// TIA Portal project "Parcial_Segundo_Corte" (V16)

(* hardware
DEVICE "S71500/ET200MP station_2"  S7-1500 station
   slot 0: "PM 190W 120/230VAC"  PM 190W 120/230VAC  6EP1333-4BA00
   slot 0: "Perfil soporte_0"  Rack  6ES7 590-1***0-0AA0
   slot 1: "MAESTRO"  CPU 1516-3 PN/DP  6ES7 516-3AN02-0AB0  V2.8
      slot 3: "Display de la CPU_1"  6ES7591-1BA00-0AA0
      slot 32768: "Interfaz PROFINET_1"  X1
         slot 32769: "Puerto_1"  X1 P1
         slot 32770: "Puerto_2"  X1 P2
      slot 33024: "Interfaz PROFINET_2"  X2
         slot 33025: "Puerto_1"  X2 P1
      slot 33280: "Interfaz DP_1"  X3
      slot 34817: "Virtual CP interface port_1"  Virtual CP interface port  Virtual CP interface port
   slot 2: "DI 32x24VDC HF_1"  DI 32x24VDC HF  6ES7 521-1BL00-0AB0  V2.0
   slot 3: "DQ 32x24VDC/0.5A ST_1"  DQ 32x24VDC/0.5A ST  6ES7 522-1BL00-0AB0  V1.0
   slot 4: "AI 8xU/I/RTD/TC ST_1"  AI 8xU/I/RTD/TC ST  6ES7 531-7KF00-0AB0  V2.0
   slot 5: "AQ 4xU/I ST_1"  AQ 4xU/I ST  6ES7 532-5HD00-0AB0  V2.0
DEVICE "S71500/ET200MP station_1"  S7-1500 station
   slot 0: "Perfil soporte_0"  Rack  6ES7 590-1***0-0AA0
   slot 0: "PM 190W 120/230VAC"  PM 190W 120/230VAC  6EP1333-4BA00
   slot 1: "ESCLAVO"  CPU 1516-3 PN/DP  6ES7 516-3AN02-0AB0  V2.8
      slot 3: "Display de la CPU_1"  6ES7591-1BA00-0AA0
      slot 32768: "Interfaz PROFINET_1"  X1
         slot 32769: "Puerto_1"  X1 P1
         slot 32770: "Puerto_2"  X1 P2
      slot 33024: "Interfaz PROFINET_2"  X2
         slot 33025: "Puerto_1"  X2 P1
      slot 33280: "Interfaz DP_1"  X3
      slot 34817: "Virtual CP interface port_1"  Virtual CP interface port  Virtual CP interface port
   slot 2: "DI 32x24VDC HF_1"  DI 32x24VDC HF  6ES7 521-1BL00-0AB0  V2.0
   slot 3: "DQ 32x24VDC/0.5A ST_1"  DQ 32x24VDC/0.5A ST  6ES7 522-1BL00-0AB0  V1.0
   slot 4: "AI 8xU/I/RTD/TC ST_1"  AI 8xU/I/RTD/TC ST  6ES7 531-7KF00-0AB0  V2.0
   slot 5: "AQ 4xU/I ST_1"  AQ 4xU/I ST  6ES7 532-5HD00-0AB0  V2.0
DEVICE "S7300/ET200M station_2"  S7-300 station
   slot 0: "Perfil soporte_0"  Rail  6ES7 390-1***0-0AA0
   slot 1: "PS 307 5A_1"  PS 307 5A  6ES7 307-1EA00-0AA0
   slot 2: "ESCLAVO_300"  CPU 314C-2 DP  6ES7 314-6CG03-0AB0  V2.6
      slot 0: "Interfaz MPI_1"  X1
      slot 1: "Interfaz DP_1"  X2
      slot 2: "DI 24/DO 16_1"  DI24/DO16
      slot 3: "AI 5/AO 2_1"  AI5/AO2
      slot 4: "Contaje_1"  Counter
      slot 5: "Posicionamiento_1"  Positioning
DEVICE "S7300/ET200M station_1"  S7-300 station
   slot 0: "Perfil soporte_0"  Rail  6ES7 390-1***0-0AA0
   slot 1: "PS 307 5A_1"  PS 307 5A  6ES7 307-1EA00-0AA0
   slot 2: "MAESTRO_300"  CPU 314C-2 DP  6ES7 314-6CG03-0AB0  V2.6
      slot 0: "Interfaz MPI_1"  X1
      slot 1: "Interfaz DP_1"  X2
      slot 2: "DI 24/DO 16_1"  DI24/DO16
      slot 3: "AI 5/AO 2_1"  AI5/AO2
      slot 4: "Contaje_1"  Counter
      slot 5: "Posicionamiento_1"  Positioning
*)

// ===== PLC "ESCLAVO"  CPU 1516-3 PN/DP =====

VAR_GLOBAL   // PLC tag table "COMUNICACION"
   "Clock_Byte" AT %MB0 : Byte;
   "Clock_10Hz" AT %M0.0 : Bool;
   "Clock_5Hz" AT %M0.1 : Bool;
   "Clock_2.5Hz" AT %M0.2 : Bool;
   "Clock_2Hz" AT %M0.3 : Bool;
   "Clock_1.25Hz" AT %M0.4 : Bool;
   "Clock_1Hz" AT %M0.5 : Bool;
   "Clock_0.625Hz" AT %M0.6 : Bool;
   "Clock_0.5Hz" AT %M0.7 : Bool;
   "Tag_1" AT %MB30 : Byte;
   "Tag_2" AT %MB40 : Byte;
   "MARCAM30.0" AT %M30.0 : Bool;
   "MARCAM30.1" AT %M30.1 : Bool;
   "MARCAM30.2" AT %M30.2 : Bool;
   "MARCAM30.3" AT %M30.3 : Bool;
   "MARCAM30.4" AT %M30.4 : Bool;
   "MARCAM30.5" AT %M30.5 : Bool;
   "MARCAM30.6" AT %M30.6 : Bool;
   "MARCAM30.7" AT %M30.7 : Bool;
   "MARCAM40.0" AT %M40.0 : Bool;
   "MARCAM40.1" AT %M40.1 : Bool;
   "MARCAM40.2" AT %M40.2 : Bool;
   "MARCAM40.3" AT %M40.3 : Bool;
   "MARCAM40.4" AT %M40.4 : Bool;
   "MARCAM40.5" AT %M40.5 : Bool;
   "MARCAM40.6" AT %M40.6 : Bool;
   "MARCAM40.7" AT %M40.7 : Bool;
   "Tag_3" AT %M200.0 : Bool;
   "Tag_4" AT %M200.1 : Bool;
   "Tag_5" AT %M200.2 : Bool;
   "Tag_6" AT %M200.3 : Bool;
   "Tag_7" AT %M200.4 : Bool;
   "Tag_8" AT %M200.5 : Bool;
   "Tag_9" AT %M200.6 : Bool;
   "Tag_10" AT %M200.7 : Bool;
   "Tag_11" AT %M300.0 : Bool;
   "Tag_12" AT %M300.1 : Bool;
   "Tag_13" AT %M300.2 : Bool;
   "Tag_14" AT %M300.4 : Bool;
   "Tag_15" AT %M300.3 : Bool;
   "Tag_16" AT %M300.5 : Bool;
   "Tag_17" AT %M300.6 : Bool;
   "Tag_18" AT %M300.7 : Bool;
END_VAR

// folder: System blocks/Program resources

DATA_BLOCK "ESCLAVO_Receive_DB"   // DB2
{ S7_Optimized_Access := 'TRUE' }
AUTHOR : SIMATIC
FAMILY : MC7Plus
NAME : TC_IP_v4
VERSION : 1.0
// stored: InstanceOfName TCON_IP_v4
"TCON_IP_v4"
BEGIN
   ID := 1;
   InterfaceId := 64;
   LocalPort := 2000;
   RemoteAddress.ADDR[1] := 192;
   RemoteAddress.ADDR[2] := 168;
   RemoteAddress.ADDR[4] := 10;
END_DATA_BLOCK

// folder: (top level)

FUNCTION "comunicacion" : Void   // FC1, LAD
{ S7_Optimized_Access := 'TRUE' }
VERSION : 0.1
BEGIN

REGION Network 1: RECIBIR ESCLAVO
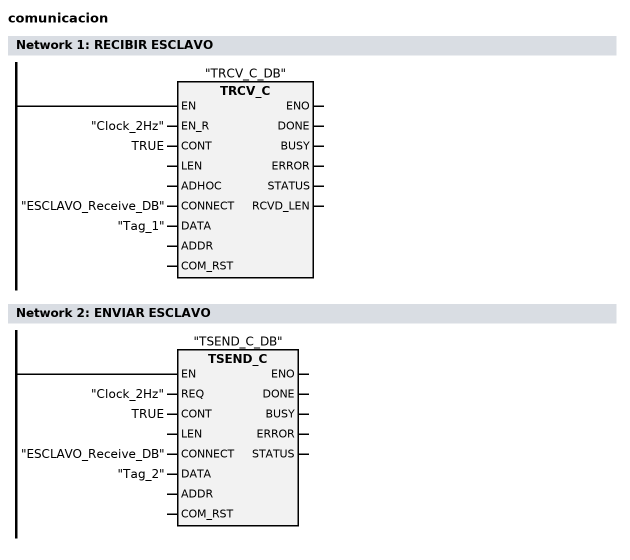
   "TRCV_C_DB"(EN_R := "Clock_2Hz", CONT := TRUE, CONNECT := "ESCLAVO_Receive_DB", DATA := "Tag_1");   // TRCV_C
END_REGION

REGION Network 2: ENVIAR ESCLAVO
   "TSEND_C_DB"(REQ := "Clock_2Hz", CONT := TRUE, CONNECT := "ESCLAVO_Receive_DB", DATA := "Tag_2");   // TSEND_C
END_REGION
END_FUNCTION

FUNCTION "compuertas" : Void   // FC2, LAD
{ S7_Optimized_Access := 'TRUE' }
VERSION : 0.1
BEGIN

REGION Network 1: SALIDAS ESCLAVO
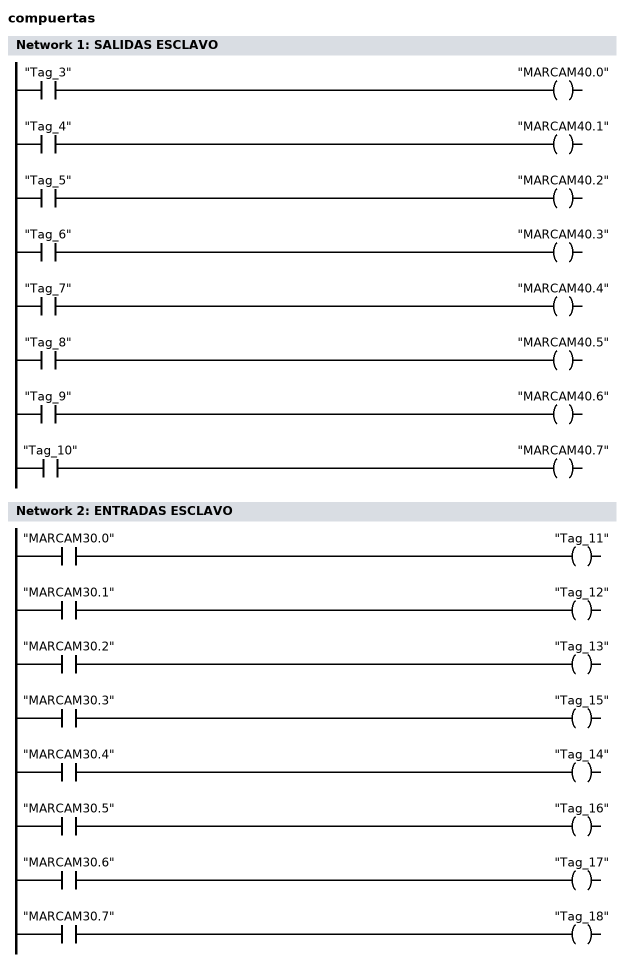
   RUNG wire#powerrail
      Contact( "Tag_3" )
      Coil( "MARCAM40.0" )
   END_RUNG
   RUNG wire#powerrail
      Contact( "Tag_4" )
      Coil( "MARCAM40.1" )
   END_RUNG
   RUNG wire#powerrail
      Contact( "Tag_5" )
      Coil( "MARCAM40.2" )
   END_RUNG
   RUNG wire#powerrail
      Contact( "Tag_6" )
      Coil( "MARCAM40.3" )
   END_RUNG
   RUNG wire#powerrail
      Contact( "Tag_7" )
      Coil( "MARCAM40.4" )
   END_RUNG
   RUNG wire#powerrail
      Contact( "Tag_8" )
      Coil( "MARCAM40.5" )
   END_RUNG
   RUNG wire#powerrail
      Contact( "Tag_9" )
      Coil( "MARCAM40.6" )
   END_RUNG
   RUNG wire#powerrail
      Contact( "Tag_10" )
      Coil( "MARCAM40.7" )
   END_RUNG
   // the same network as SCL:
   "MARCAM40.0" := "Tag_3";
   "MARCAM40.1" := "Tag_4";
   "MARCAM40.2" := "Tag_5";
   "MARCAM40.3" := "Tag_6";
   "MARCAM40.4" := "Tag_7";
   "MARCAM40.5" := "Tag_8";
   "MARCAM40.6" := "Tag_9";
   "MARCAM40.7" := "Tag_10";
END_REGION

REGION Network 2: ENTRADAS ESCLAVO
   RUNG wire#powerrail
      Contact( "MARCAM30.0" )
      Coil( "Tag_11" )
   END_RUNG
   RUNG wire#powerrail
      Contact( "MARCAM30.1" )
      Coil( "Tag_12" )
   END_RUNG
   RUNG wire#powerrail
      Contact( "MARCAM30.2" )
      Coil( "Tag_13" )
   END_RUNG
   RUNG wire#powerrail
      Contact( "MARCAM30.3" )
      Coil( "Tag_15" )
   END_RUNG
   RUNG wire#powerrail
      Contact( "MARCAM30.4" )
      Coil( "Tag_14" )
   END_RUNG
   RUNG wire#powerrail
      Contact( "MARCAM30.5" )
      Coil( "Tag_16" )
   END_RUNG
   RUNG wire#powerrail
      Contact( "MARCAM30.6" )
      Coil( "Tag_17" )
   END_RUNG
   RUNG wire#powerrail
      Contact( "MARCAM30.7" )
      Coil( "Tag_18" )
   END_RUNG
   // the same network as SCL:
   "Tag_11" := "MARCAM30.0";
   "Tag_12" := "MARCAM30.1";
   "Tag_13" := "MARCAM30.2";
   "Tag_15" := "MARCAM30.3";
   "Tag_14" := "MARCAM30.4";
   "Tag_16" := "MARCAM30.5";
   "Tag_17" := "MARCAM30.6";
   "Tag_18" := "MARCAM30.7";
END_REGION
END_FUNCTION

ORGANIZATION_BLOCK "Main"   // OB1, LAD, ProgramCycle
TITLE = "Main Program Sweep (Cycle)"
{ S7_Optimized_Access := 'TRUE' }
VERSION : 0.1
   VAR_INPUT
      Initial_Call : Bool;   // Initial call of this OB
      Remanence : Bool;   // =True, if remanent data are available
   END_VAR
BEGIN

REGION Network 1: COMUNICACION ETHERNET
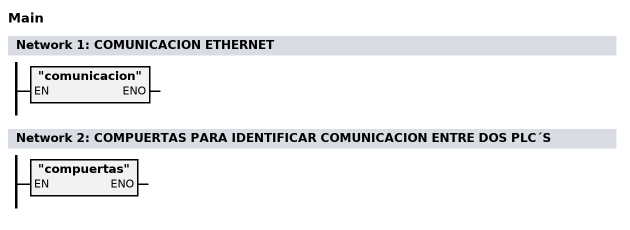
   RUNG wire#powerrail
      "comunicacion"()
   END_RUNG
   // the same network as SCL:
   "comunicacion"();
END_REGION

REGION Network 2: COMPUERTAS PARA IDENTIFICAR COMUNICACION ENTRE DOS PLC´S
   RUNG wire#powerrail
      "compuertas"()
   END_RUNG
   // the same network as SCL:
   "compuertas"();
END_REGION
END_ORGANIZATION_BLOCK

// ===== PLC "MAESTRO"  CPU 1516-3 PN/DP =====

VAR_GLOBAL   // PLC tag table "COMUNICACION"
   "Clock_Byte" AT %MB0 : Byte;
   "Clock_10Hz" AT %M0.0 : Bool;
   "Clock_5Hz" AT %M0.1 : Bool;
   "Clock_2.5Hz" AT %M0.2 : Bool;
   "Clock_2Hz" AT %M0.3 : Bool;
   "Clock_1.25Hz" AT %M0.4 : Bool;
   "Clock_1Hz" AT %M0.5 : Bool;
   "Clock_0.625Hz" AT %M0.6 : Bool;
   "Clock_0.5Hz" AT %M0.7 : Bool;
   "Tag_1" AT %MB20 : Byte;
   "Tag_2" AT %MB50 : Byte;
   "MARCAM20.0" AT %M20.0 : Bool;
   "MARCAM20.1" AT %M20.1 : Bool;
   "MARCAM20.2" AT %M20.2 : Bool;
   "MARCAM20.3" AT %M20.3 : Bool;
   "MARCAM20.4" AT %M20.4 : Bool;
   "MARCAM20.5" AT %M20.5 : Bool;
   "MARCAM20.6" AT %M20.6 : Bool;
   "MARCAM20.7" AT %M20.7 : Bool;
   "MARCAM50.0" AT %M50.0 : Bool;
   "MARCAM50.1" AT %M50.1 : Bool;
   "MARCAM50.2" AT %M50.2 : Bool;
   "MARCAM50.3" AT %M50.3 : Bool;
   "MARCAM50.4" AT %M50.4 : Bool;
   "MARCAM50.5" AT %M50.5 : Bool;
   "MARCAM50.6" AT %M50.6 : Bool;
   "MARCAM50.7" AT %M50.7 : Bool;
   "Tag_3" AT %M100.0 : Bool;
   "Tag_4" AT %M100.1 : Bool;
   "Tag_5" AT %M100.2 : Bool;
   "Tag_6" AT %M100.3 : Bool;
   "Tag_7" AT %M100.4 : Bool;
   "Tag_8" AT %M100.5 : Bool;
   "Tag_9" AT %M100.6 : Bool;
   "Tag_10" AT %M100.7 : Bool;
   "Tag_11" AT %M300.0 : Bool;
   "Tag_12" AT %M300.1 : Bool;
   "Tag_13" AT %M300.2 : Bool;
   "Tag_14" AT %M300.3 : Bool;
   "Tag_15" AT %M300.4 : Bool;
   "Tag_16" AT %M300.5 : Bool;
   "Tag_17" AT %M300.6 : Bool;
   "Tag_18" AT %M300.7 : Bool;
END_VAR

// folder: System blocks/Program resources

DATA_BLOCK "MAESTRO_Send_DB"   // DB2
{ S7_Optimized_Access := 'TRUE' }
AUTHOR : SIMATIC
FAMILY : MC7Plus
NAME : TC_IP_v4
VERSION : 1.0
// stored: InstanceOfName TCON_IP_v4
"TCON_IP_v4"
BEGIN
   ID := 1;
   InterfaceId := 64;
   RemotePort := 2000;
   ActiveEstablished := true;
   RemoteAddress.ADDR[1] := 192;
   RemoteAddress.ADDR[2] := 168;
   RemoteAddress.ADDR[4] := 20;
END_DATA_BLOCK

// folder: (top level)

FUNCTION "comunicacion" : Void   // FC1, LAD
{ S7_Optimized_Access := 'TRUE' }
VERSION : 0.1
BEGIN

REGION Network 1: ENVIAR MAESTRO
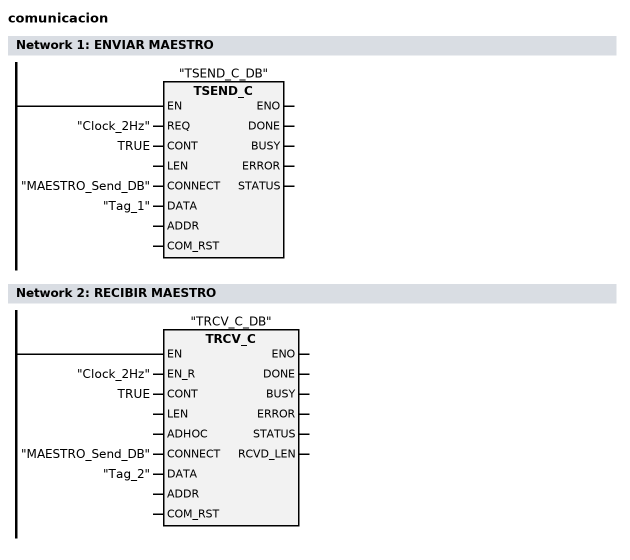
   "TSEND_C_DB"(REQ := "Clock_2Hz", CONT := TRUE, CONNECT := "MAESTRO_Send_DB", DATA := "Tag_1");   // TSEND_C
END_REGION

REGION Network 2: RECIBIR MAESTRO
   "TRCV_C_DB"(EN_R := "Clock_2Hz", CONT := TRUE, CONNECT := "MAESTRO_Send_DB", DATA := "Tag_2");   // TRCV_C
END_REGION
END_FUNCTION

FUNCTION "Compuertas" : Void   // FC2, LAD
{ S7_Optimized_Access := 'TRUE' }
VERSION : 0.1
BEGIN

REGION Network 1: SALIDAS MAESTRO
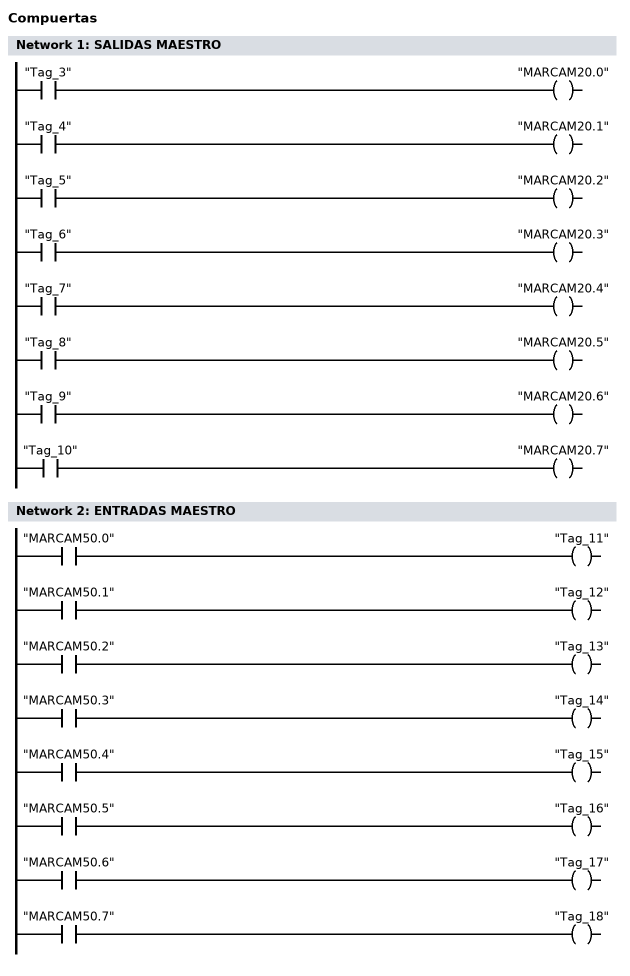
   RUNG wire#powerrail
      Contact( "Tag_3" )
      Coil( "MARCAM20.0" )
   END_RUNG
   RUNG wire#powerrail
      Contact( "Tag_4" )
      Coil( "MARCAM20.1" )
   END_RUNG
   RUNG wire#powerrail
      Contact( "Tag_5" )
      Coil( "MARCAM20.2" )
   END_RUNG
   RUNG wire#powerrail
      Contact( "Tag_6" )
      Coil( "MARCAM20.3" )
   END_RUNG
   RUNG wire#powerrail
      Contact( "Tag_7" )
      Coil( "MARCAM20.4" )
   END_RUNG
   RUNG wire#powerrail
      Contact( "Tag_8" )
      Coil( "MARCAM20.5" )
   END_RUNG
   RUNG wire#powerrail
      Contact( "Tag_9" )
      Coil( "MARCAM20.6" )
   END_RUNG
   RUNG wire#powerrail
      Contact( "Tag_10" )
      Coil( "MARCAM20.7" )
   END_RUNG
   // the same network as SCL:
   "MARCAM20.0" := "Tag_3";
   "MARCAM20.1" := "Tag_4";
   "MARCAM20.2" := "Tag_5";
   "MARCAM20.3" := "Tag_6";
   "MARCAM20.4" := "Tag_7";
   "MARCAM20.5" := "Tag_8";
   "MARCAM20.6" := "Tag_9";
   "MARCAM20.7" := "Tag_10";
END_REGION

REGION Network 2: ENTRADAS MAESTRO
   RUNG wire#powerrail
      Contact( "MARCAM50.0" )
      Coil( "Tag_11" )
   END_RUNG
   RUNG wire#powerrail
      Contact( "MARCAM50.1" )
      Coil( "Tag_12" )
   END_RUNG
   RUNG wire#powerrail
      Contact( "MARCAM50.2" )
      Coil( "Tag_13" )
   END_RUNG
   RUNG wire#powerrail
      Contact( "MARCAM50.3" )
      Coil( "Tag_14" )
   END_RUNG
   RUNG wire#powerrail
      Contact( "MARCAM50.4" )
      Coil( "Tag_15" )
   END_RUNG
   RUNG wire#powerrail
      Contact( "MARCAM50.5" )
      Coil( "Tag_16" )
   END_RUNG
   RUNG wire#powerrail
      Contact( "MARCAM50.6" )
      Coil( "Tag_17" )
   END_RUNG
   RUNG wire#powerrail
      Contact( "MARCAM50.7" )
      Coil( "Tag_18" )
   END_RUNG
   // the same network as SCL:
   "Tag_11" := "MARCAM50.0";
   "Tag_12" := "MARCAM50.1";
   "Tag_13" := "MARCAM50.2";
   "Tag_14" := "MARCAM50.3";
   "Tag_15" := "MARCAM50.4";
   "Tag_16" := "MARCAM50.5";
   "Tag_17" := "MARCAM50.6";
   "Tag_18" := "MARCAM50.7";
END_REGION
END_FUNCTION

ORGANIZATION_BLOCK "Main"   // OB1, LAD, ProgramCycle
TITLE = "Main Program Sweep (Cycle)"
{ S7_Optimized_Access := 'TRUE' }
VERSION : 0.1
   VAR_INPUT
      Initial_Call : Bool;   // Initial call of this OB
      Remanence : Bool;   // =True, if remanent data are available
   END_VAR
BEGIN

REGION Network 1
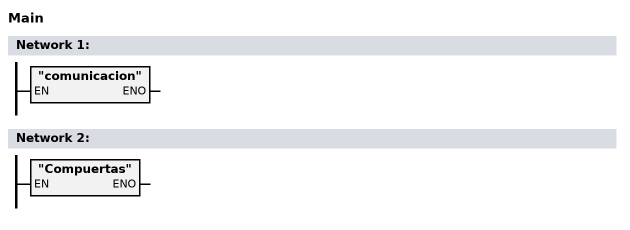
   RUNG wire#powerrail
      "comunicacion"()
   END_RUNG
   // the same network as SCL:
   "comunicacion"();
END_REGION

REGION Network 2
   RUNG wire#powerrail
      "Compuertas"()
   END_RUNG
   // the same network as SCL:
   "Compuertas"();
END_REGION
END_ORGANIZATION_BLOCK

// ===== PLC "MAESTRO_300"  CPU 314C-2 DP =====

VAR_GLOBAL   // PLC tag table "Tabla de variables estándar"
   "ENVIAR_DATO" AT %MB0 : Byte;
   "DATO_ENVIADO" AT %QB120 : Byte;
   "DATO_RECIBIDO" AT %IB240 : Byte;
   "VISUALIZAR_DATO" AT %MB3 : Byte;
END_VAR

FUNCTION "comunicacion" : Void   // FC1, LAD
{ S7_Optimized_Access := 'FALSE' }
VERSION : 0.1
BEGIN

REGION Network 1
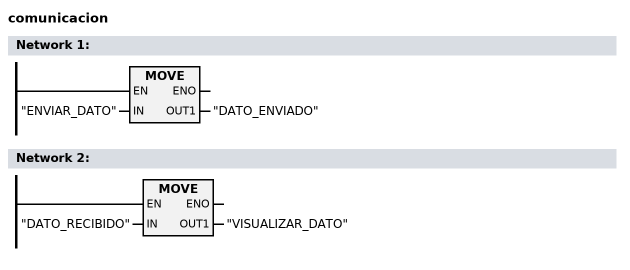
   RUNG wire#powerrail
      { S7_GenerateENO := "TRUE" } Move(in := "ENVIAR_DATO", out1 => "DATO_ENVIADO")
   END_RUNG
   // the same network as SCL:
   "DATO_ENVIADO" := "ENVIAR_DATO";
END_REGION

REGION Network 2
   RUNG wire#powerrail
      { S7_GenerateENO := "TRUE" } Move(in := "DATO_RECIBIDO", out1 => "VISUALIZAR_DATO")
   END_RUNG
   // the same network as SCL:
   "VISUALIZAR_DATO" := "DATO_RECIBIDO";
END_REGION
END_FUNCTION

ORGANIZATION_BLOCK "Main"   // OB1, LAD
TITLE = "Main Program Sweep (Cycle)"
{ S7_Optimized_Access := 'FALSE' }
VERSION : 0.1
   VAR_TEMP
      OB1_EV_CLASS : Byte;   // Bits 0-3 = 1 (Coming event), Bits 4-7 = 1 (Event class 1)
      OB1_SCAN_1 : Byte;   // 1 (Cold restart scan 1 of OB 1), 3 (Scan 2-n of OB 1)
      OB1_PRIORITY : Byte;   // Priority of OB Execution
      OB1_OB_NUMBR : Byte;   // 1 (Organization block 1, OB1)
      OB1_RESERVED_1 : Byte;   // Reserved for system
      OB1_RESERVED_2 : Byte;   // Reserved for system
      OB1_PREV_CYCLE : Int;   // Cycle time of previous OB1 scan (milliseconds)
      OB1_MIN_CYCLE : Int;   // Minimum cycle time of OB1 (milliseconds)
      OB1_MAX_CYCLE : Int;   // Maximum cycle time of OB1 (milliseconds)
      OB1_DATE_TIME : Date_And_Time;   // Date and time OB1 started
   END_VAR
BEGIN

REGION Network 1
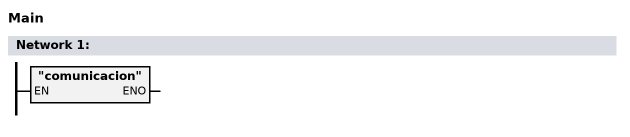
   RUNG wire#powerrail
      "comunicacion"()
   END_RUNG
   // the same network as SCL:
   "comunicacion"();
END_REGION
END_ORGANIZATION_BLOCK

ORGANIZATION_BLOCK "I/O_FLT1"   // OB82, FBD
TITLE = "I/O Point Fault"
{ S7_Optimized_Access := 'FALSE' }
VERSION : 0.1
   VAR_TEMP
      OB82_EV_CLASS : Byte;   // 16#39, Event class 3, Entering event state, Internal fault event
      OB82_FLT_ID : Byte;   // 16#XX, Fault identifcation code
      OB82_PRIORITY : Byte;   // Priority of OB Execution
      OB82_OB_NUMBR : Byte;   // 82 (Organization block 82, OB82)
      OB82_RESERVED_1 : Byte;   // Reserved for system
      OB82_IO_FLAG : Byte;   // Input (01010100), Output (01010101)
      OB82_MDL_ADDR : Word;   // Base address of module with fault
      OB82_MDL_DEFECT : Bool;   // Module defective
      OB82_INT_FAULT : Bool;   // Internal fault
      OB82_EXT_FAULT : Bool;   // External fault
      OB82_PNT_INFO : Bool;   // Point information
      OB82_EXT_VOLTAGE : Bool;   // External voltage low
      OB82_FLD_CONNCTR : Bool;   // Field wiring connector missing
      OB82_NO_CONFIG : Bool;   // Module has no configuration data
      OB82_CONFIG_ERR : Bool;   // Module has configuration error
      OB82_MDL_TYPE : Byte;   // Type of module
      OB82_SUB_MDL_ERR : Bool;   // Sub-Module is missing or has error
      OB82_COMM_FAULT : Bool;   // Communication fault
      OB82_MDL_STOP : Bool;   // Module is stopped
      OB82_WTCH_DOG_FLT : Bool;   // Watch dog timer stopped module
      OB82_INT_PS_FLT : Bool;   // Internal power supply fault
      OB82_PRIM_BATT_FLT : Bool;   // Primary battery is in fault
      OB82_BCKUP_BATT_FLT : Bool;   // Backup battery is in fault
      OB82_RESERVED_2 : Bool;   // Reserved for system
      OB82_RACK_FLT : Bool;   // Rack fault, only for bus interface module
      OB82_PROC_FLT : Bool;   // Processor fault
      OB82_EPROM_FLT : Bool;   // EPROM fault
      OB82_RAM_FLT : Bool;   // RAM fault
      OB82_ADU_FLT : Bool;   // ADU fault
      OB82_FUSE_FLT : Bool;   // Fuse fault
      OB82_HW_INTR_FLT : Bool;   // Hardware interupt input in fault
      OB82_RESERVED_3 : Bool;   // Reserved for system
      OB82_DATE_TIME : Date_And_Time;   // Date and time OB82 started
   END_VAR
BEGIN
END_ORGANIZATION_BLOCK

ORGANIZATION_BLOCK "RACK_FLT"   // OB86, FBD
TITLE = "Loss Of Rack Fault"
{ S7_Optimized_Access := 'FALSE' }
VERSION : 0.1
   VAR_TEMP
      OB86_EV_CLASS : Byte;   // 16#38/39 Event class 3
      OB86_FLT_ID : Byte;   // 16#C1/C4/C5, Fault identification code
      OB86_PRIORITY : Byte;   // Priority of OB Execution
      OB86_OB_NUMBR : Byte;   // 86 (Organization block 86, OB86)
      OB86_RESERVED_1 : Byte;   // Reserved for system
      OB86_RESERVED_2 : Byte;   // Reserved for system
      OB86_MDL_ADDR : Word;   // Base address of IM module in rack with fault
      OB86_RACKS_FLTD : Array[0..31] of Bool;   // Racks in fault
      OB86_DATE_TIME : Date_And_Time;   // Date and time OB86 started
   END_VAR
BEGIN
END_ORGANIZATION_BLOCK

// ===== PLC "ESCLAVO_300"  CPU 314C-2 DP =====

VAR_GLOBAL   // PLC tag table "Tabla de variables estándar"
   "ENVIAR_DATO" AT %MB0 : Byte;
   "DATO_ENVIADO" AT %QB240 : Byte;
   "DATO_RECIBIDO" AT %IB120 : Byte;
   "VISUALIZAR_DATO" AT %MB4 : Byte;
END_VAR

FUNCTION "comunicacion" : Void   // FC1, LAD
{ S7_Optimized_Access := 'FALSE' }
VERSION : 0.1
BEGIN

REGION Network 1
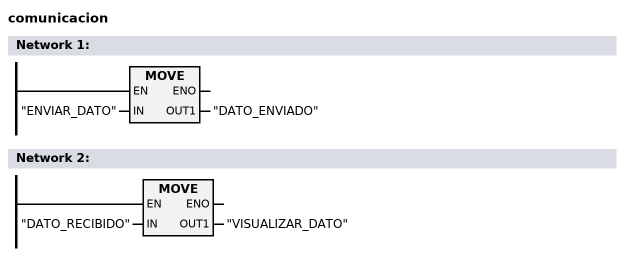
   RUNG wire#powerrail
      { S7_GenerateENO := "TRUE" } Move(in := "ENVIAR_DATO", out1 => "DATO_ENVIADO")
   END_RUNG
   // the same network as SCL:
   "DATO_ENVIADO" := "ENVIAR_DATO";
END_REGION

REGION Network 2
   RUNG wire#powerrail
      { S7_GenerateENO := "TRUE" } Move(in := "DATO_RECIBIDO", out1 => "VISUALIZAR_DATO")
   END_RUNG
   // the same network as SCL:
   "VISUALIZAR_DATO" := "DATO_RECIBIDO";
END_REGION
END_FUNCTION

ORGANIZATION_BLOCK "Main"   // OB1, LAD
TITLE = "Main Program Sweep (Cycle)"
{ S7_Optimized_Access := 'FALSE' }
VERSION : 0.1
   VAR_TEMP
      OB1_EV_CLASS : Byte;   // Bits 0-3 = 1 (Coming event), Bits 4-7 = 1 (Event class 1)
      OB1_SCAN_1 : Byte;   // 1 (Cold restart scan 1 of OB 1), 3 (Scan 2-n of OB 1)
      OB1_PRIORITY : Byte;   // Priority of OB Execution
      OB1_OB_NUMBR : Byte;   // 1 (Organization block 1, OB1)
      OB1_RESERVED_1 : Byte;   // Reserved for system
      OB1_RESERVED_2 : Byte;   // Reserved for system
      OB1_PREV_CYCLE : Int;   // Cycle time of previous OB1 scan (milliseconds)
      OB1_MIN_CYCLE : Int;   // Minimum cycle time of OB1 (milliseconds)
      OB1_MAX_CYCLE : Int;   // Maximum cycle time of OB1 (milliseconds)
      OB1_DATE_TIME : Date_And_Time;   // Date and time OB1 started
   END_VAR
BEGIN

REGION Network 1
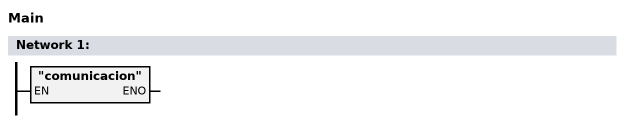
   RUNG wire#powerrail
      "comunicacion"()
   END_RUNG
   // the same network as SCL:
   "comunicacion"();
END_REGION
END_ORGANIZATION_BLOCK

ORGANIZATION_BLOCK "I/O_FLT1"   // OB82, FBD
TITLE = "I/O Point Fault"
{ S7_Optimized_Access := 'FALSE' }
VERSION : 0.1
   VAR_TEMP
      OB82_EV_CLASS : Byte;   // 16#39, Event class 3, Entering event state, Internal fault event
      OB82_FLT_ID : Byte;   // 16#XX, Fault identifcation code
      OB82_PRIORITY : Byte;   // Priority of OB Execution
      OB82_OB_NUMBR : Byte;   // 82 (Organization block 82, OB82)
      OB82_RESERVED_1 : Byte;   // Reserved for system
      OB82_IO_FLAG : Byte;   // Input (01010100), Output (01010101)
      OB82_MDL_ADDR : Word;   // Base address of module with fault
      OB82_MDL_DEFECT : Bool;   // Module defective
      OB82_INT_FAULT : Bool;   // Internal fault
      OB82_EXT_FAULT : Bool;   // External fault
      OB82_PNT_INFO : Bool;   // Point information
      OB82_EXT_VOLTAGE : Bool;   // External voltage low
      OB82_FLD_CONNCTR : Bool;   // Field wiring connector missing
      OB82_NO_CONFIG : Bool;   // Module has no configuration data
      OB82_CONFIG_ERR : Bool;   // Module has configuration error
      OB82_MDL_TYPE : Byte;   // Type of module
      OB82_SUB_MDL_ERR : Bool;   // Sub-Module is missing or has error
      OB82_COMM_FAULT : Bool;   // Communication fault
      OB82_MDL_STOP : Bool;   // Module is stopped
      OB82_WTCH_DOG_FLT : Bool;   // Watch dog timer stopped module
      OB82_INT_PS_FLT : Bool;   // Internal power supply fault
      OB82_PRIM_BATT_FLT : Bool;   // Primary battery is in fault
      OB82_BCKUP_BATT_FLT : Bool;   // Backup battery is in fault
      OB82_RESERVED_2 : Bool;   // Reserved for system
      OB82_RACK_FLT : Bool;   // Rack fault, only for bus interface module
      OB82_PROC_FLT : Bool;   // Processor fault
      OB82_EPROM_FLT : Bool;   // EPROM fault
      OB82_RAM_FLT : Bool;   // RAM fault
      OB82_ADU_FLT : Bool;   // ADU fault
      OB82_FUSE_FLT : Bool;   // Fuse fault
      OB82_HW_INTR_FLT : Bool;   // Hardware interupt input in fault
      OB82_RESERVED_3 : Bool;   // Reserved for system
      OB82_DATE_TIME : Date_And_Time;   // Date and time OB82 started
   END_VAR
BEGIN
END_ORGANIZATION_BLOCK

ORGANIZATION_BLOCK "RACK_FLT"   // OB86, FBD
TITLE = "Loss Of Rack Fault"
{ S7_Optimized_Access := 'FALSE' }
VERSION : 0.1
   VAR_TEMP
      OB86_EV_CLASS : Byte;   // 16#38/39 Event class 3
      OB86_FLT_ID : Byte;   // 16#C1/C4/C5, Fault identification code
      OB86_PRIORITY : Byte;   // Priority of OB Execution
      OB86_OB_NUMBR : Byte;   // 86 (Organization block 86, OB86)
      OB86_RESERVED_1 : Byte;   // Reserved for system
      OB86_RESERVED_2 : Byte;   // Reserved for system
      OB86_MDL_ADDR : Word;   // Base address of IM module in rack with fault
      OB86_RACKS_FLTD : Array[0..31] of Bool;   // Racks in fault
      OB86_DATE_TIME : Date_And_Time;   // Date and time OB86 started
   END_VAR
BEGIN
END_ORGANIZATION_BLOCK